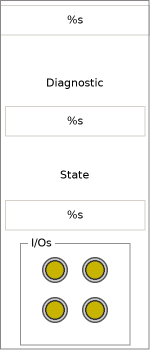
VISUALIZATION DiagConnELx904  // 150x350
VAR_INPUT
	connName:STRING(20);
	diag:E_connInfoDiag;
	state:STRING(20);
	bits:ARRAY[0..3] OF BOOL;
END_VAR
    GroupBox (20,235 110x110), "I/Os"
        Lamp1 (20,20 30x30), variable: bits[0], style: Lamp-Lamp1-Yellow
        Lamp1 (60,20 30x30), variable: bits[2], style: Lamp-Lamp1-Yellow
        Lamp1 (20,60 30x30), variable: bits[1], style: Lamp-Lamp1-Yellow
        Lamp1 (60,60 30x30), variable: bits[3], style: Lamp-Lamp1-Yellow
    Label (5,68 140x30), "Diagnostic"
    Label (5,160 140x30), "State"
    Textfield (5,106 140x30), "%s", text variable: diag
    Textfield (5,200 140x30), "%s", text variable: state
    Textfield (0,5 150x30), "%s", text variable: connName
END_VISUALIZATION

(* stored: Version 1.1.0.1, ProductVersion 3.1.4024.12
   Visu DiagConnELx904: Id {41f85d8a-7324-4b8c-8d14-439381896ae6} *)
